FUNCTION_BLOCK IO_DQ32_HMI (* Service Interface Function Block Type *)
  (* Standard: 61499-2 *)
  (* Version 0.0, 10/2/2026, Schneider Electric, template *)
  PACKAGE Hidryco.HidrycoLib;
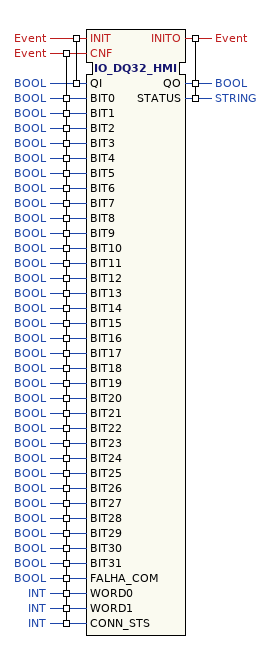
  EVENT_INPUT
    INIT WITH QI;
    CNF WITH BIT0, BIT1, BIT2, BIT3, BIT4, BIT5, BIT6, BIT7, BIT8, BIT9, BIT10, BIT11, BIT12, BIT13, BIT14, BIT15, BIT16, BIT17, BIT18, BIT19, BIT20, BIT21, BIT22, BIT23, BIT24, BIT25, BIT26, BIT27, BIT28, BIT29, BIT30, BIT31, FALHA_COM, WORD0, WORD1, CONN_STS; (* Atualiza o depurador *)
  END_EVENT
  EVENT_OUTPUT
    INITO WITH QO, STATUS;
  END_EVENT
  VAR_INPUT
    QI : BOOL;
    BIT0 : BOOL; (* DO 0 *)
    BIT1 : BOOL; (* DO 1 *)
    BIT2 : BOOL; (* DO 2 *)
    BIT3 : BOOL; (* DO 3 *)
    BIT4 : BOOL; (* DO 4 *)
    BIT5 : BOOL; (* DO 5 *)
    BIT6 : BOOL; (* DO 6 *)
    BIT7 : BOOL; (* DO 7 *)
    BIT8 : BOOL; (* DO 8 *)
    BIT9 : BOOL; (* DO 9 *)
    BIT10 : BOOL; (* DO 10 *)
    BIT11 : BOOL; (* DO 11 *)
    BIT12 : BOOL; (* DO 12 *)
    BIT13 : BOOL; (* DO 13 *)
    BIT14 : BOOL; (* DO 14 *)
    BIT15 : BOOL; (* DO 15 *)
    BIT16 : BOOL; (* DO 16 *)
    BIT17 : BOOL; (* DO 17 *)
    BIT18 : BOOL; (* DO 18 *)
    BIT19 : BOOL; (* DO 19 *)
    BIT20 : BOOL; (* DO 20 *)
    BIT21 : BOOL; (* DO 21 *)
    BIT22 : BOOL; (* DO 22 *)
    BIT23 : BOOL; (* DO 23 *)
    BIT24 : BOOL; (* DO 24 *)
    BIT25 : BOOL; (* DO 25 *)
    BIT26 : BOOL; (* DO 26 *)
    BIT27 : BOOL; (* DO 27 *)
    BIT28 : BOOL; (* DO 28 *)
    BIT29 : BOOL; (* DO 29 *)
    BIT30 : BOOL; (* DO 30 *)
    BIT31 : BOOL; (* DO 31 *)
    FALHA_COM : BOOL; (* TRUE = remota offline *)
    WORD0 : INT; (* Word 0 (bits 0-15) *)
    WORD1 : INT; (* Word 1 (bits 16-31) *)
    CONN_STS : INT; (* connStatusInt: 1 online, 0 offline *)
  END_VAR
  VAR_OUTPUT
    QO : BOOL; (* Event Output Qualifier *)
    STATUS : STRING; (* Service Status *)
  END_VAR
  SERVICE /
    SEQUENCE 
    END_SEQUENCE
  END_SERVICE
END_FUNCTION_BLOCK
